(* CODESYS project StateMachineExport.export

Project tree, tasks and I/O mapping:
  program Main [ST]: HandleErrorState, HandleInitState, HandleRunState, HandleStopState
  function block StateMachineHandler [ST]: UpdateState, CurrentState, LastState
*)

// Main
PROGRAM Main
VAR
	scanCount : INT;
	
	StateHandler : StateMachineHandler;
	state : (Init, Run, Stop, Error);
END_VAR


state := StateHandler.CurrentState;

CASE StateHandler.CurrentState OF
	
	Init: HandleInitState();
	
	Run: HandleRunState();
	
	Stop: HandleStopState();
	
	Error: HandleErrorState();
	
END_CASE

scanCount := scanCount+1;

METHOD PRIVATE HandleErrorState : BOOL
VAR_INPUT
END_VAR
END_METHOD

METHOD PRIVATE HandleInitState : BOOL

IF scanCount >= 200 THEN
	scanCount := 0;
	StateHandler.UpdateState(Run);
END_IF
END_METHOD

METHOD PRIVATE HandleRunState : BOOL

IF scanCount >= 200 THEN
	scanCount := 0;
	StateHandler.UpdateState(Stop);
END_IF
END_METHOD

METHOD PRIVATE HandleStopState : BOOL

IF scanCount >= 200 THEN
	scanCount := 0;
	StateHandler.UpdateState(Init);
END_IF
END_METHOD

END_PROGRAM

// StateMachineHandler
FUNCTION_BLOCK StateMachineHandler
VAR
	_currentState : INT;
	_lastState : INT;
END_VAR

METHOD PUBLIC UpdateState : BOOL
VAR_INPUT
	requestedState : INT;
END_VAR

IF requestedState <> _currentState THEN
	_lastState := _currentState;
	_currentState := requestedState;
END_IF
END_METHOD

PROPERTY PUBLIC CurrentState : INT
GET

CurrentState := _currentState;
END_GET
END_PROPERTY

PROPERTY PUBLIC LastState : INT
GET

LastState := _lastState;
END_GET
END_PROPERTY

END_FUNCTION_BLOCK
